FUNCTION F_Scaling : DINT
VAR_INPUT
	diInput 	: DINT;
	diRef100 	: DINT;
END_VAR


VAR
END_VAR
(*All VAR_IN_OUT variables have been moved to the end of the declaration due to compatibility reasons*)
VAR_IN_OUT
	stScal 		: ST_AnalogScaling;
END_VAR

F_Scaling :=
		(diInput
		- stScal.diXRef)
	* stScal.diFact
	/ diRef100
	+ stScal.diYRef;

END_FUNCTION

(* stored: Version 1.1.0.1, ProductVersion 3.1.4018.5
   POU F_Scaling: Id {9bf93847-492f-4c8d-a970-417d937fd889}, SpecialFunc None *)
